FUNCTION_BLOCK ScreenBase EXTENDS TExecution IMPLEMENTS IDevice
VAR_INPUT
END_VAR
VAR_OUTPUT
END_VAR
VAR
	{attribute 'OPC.UA.DA' := '0'}
	_name : STRING;
	{attribute 'OPC.UA.DA' := '0'}
	_deviceID : STRING;				
	{attribute 'OPC.UA.DA' := '0'}	
	_family : DeviceFamily;	
	{attribute 'OPC.UA.DA' := '0'}
	_logger : Logger;
	{attribute 'OPC.UA.DA' := '0'}
	_message : StringBuilder;
	{attribute 'OPC.UA.DA' := '0'}
	_screenConfig : DeviceConfiguration;	
END_VAR

PROPERTY DeviceID : STRING
GET
DeviceID := _deviceID;
END_GET
SET
_deviceID := DeviceID;
END_SET
END_PROPERTY

PROPERTY Family : DeviceFamily
GET
Family := _family;
END_GET
SET
_family := Family;
END_SET
END_PROPERTY

PROPERTY Name : STRING
GET
Name := _name;
END_GET
SET
_name := Name;
END_SET
END_PROPERTY

END_FUNCTION_BLOCK

(* stored: Version 1.1.0.1, ProductVersion 3.1.4024.12
   POU ScreenBase: Id {ddf188ec-7c6d-46b8-8b21-7b6c704db19f}, SpecialFunc None
   Property DeviceID: Id {8b804620-5b32-4e4d-b7ce-4b0cdc03d87c}
   Get Get: Id {a0df453b-361e-453d-89a9-87ae9d530b6c}
   Set Set: Id {f5a38261-872d-4f16-81b6-1488ec96470b}
   Property Family: Id {89e6b0e7-ce5b-43e9-a482-661fd1cf4877}
   Get Get: Id {ed083076-6851-485b-a2e0-b5024663ae41}
   Set Set: Id {646f8f5d-828e-4325-96c9-f057d1cf5074}
   Property Name: Id {f8b33eb0-4825-40fc-bcc4-5acc7a65673d}
   Get Get: Id {3c61145f-7a0c-4bb0-a831-79f83b2264d6}
   Set Set: Id {ab54629d-ad66-4f18-84ed-3af1c2940a74} *)
